PROGRAM CheckConfig
VAR_INPUT
		IN_Start				: BOOL := TRUE;
		ParamInitWait			: TIME := T#5S;
END_VAR
VAR_OUTPUT
		OUT_aDBConfig         		: ARRAY[0..MAX_CONFIGURATIONS] OF ST_ConfigDB;
		OUT_Busy					: BOOL;
		OUT_Error					: BOOL;
		OUT_Result					: INT;
END_VAR
VAR
	// CheckConfig    
		TON_CheckConfig				: TON;      		
		TrigCheckConfig				: R_TRIG;
		TrigInit					: F_TRIG;
		RS_CheckConfig				: RS;
		                    		
		ConfigTcDBSrvEvt  			: FB_ConfigTcDBSrvEvt(sNetId := '', tTimeout:=T#5S);
		                    		
		aAutoGrpConfig    			: ARRAY[0..MAX_CONFIGURATIONS] OF ST_ConfigAutoLogGrp;
		AX_NameBase					: ARRAY[0..MAX_CONFIGURATIONS] OF T_MaxString;
		AX_hDBID					: ARRAY[0..MAX_CONFIGURATIONS] OF BOOL;
		AX_hDBIDNull				: ARRAY[0..MAX_CONFIGURATIONS] OF BOOL;
		                    		
		nDbCount          			: UDINT;
		nAutoGrpCount     			: UDINT;

		KK : UDINT;
END_VAR

TON_CheckConfig(IN := IN_Start, PT := ParamInitWait);

TrigCheckConfig(CLK := TON_CheckConfig.Q);
RS_CheckConfig(SET := TrigCheckConfig.Q);
IF TrigCheckConfig.Q THEN
	IN_Start := FALSE;
	OUT_Result := 0;
END_IF
IF RS_CheckConfig.Q1 THEN
	
	OUT_Busy := TRUE;
	IF ConfigTcDBSrvEvt.Read(pDBConfig := ADR(OUT_aDBConfig), cbDBConfig := SIZEOF(OUT_aDBConfig), pAutologGrpConfig := ADR(aAutoGrpConfig),
			cbAutoLogGrpConfig := SIZEOF(aAutoGrpConfig),pDBCount := ADR(nDbCount),pAutoLogGrpCount := ADR(nAutoGrpCount)) THEN
		
		IF ConfigTcDBSrvEvt.bError THEN
			OUT_Result := -1;
		ELSE
			FOR KK := 0 TO MAX_CONFIGURATIONS DO
				AX_hDBID[OUT_aDBConfig[KK].hDBID] := OUT_aDBConfig[KK].hDBID <> 0;
				AX_NameBase[KK] :=  OUT_aDBConfig[KK].sName;
			END_FOR
			OUT_Result := 1;
		END_IF  
		RS_CheckConfig(RESET1 := TRUE);
		RS_CheckConfig(RESET1 := FALSE);
		OUT_Busy := FALSE;
		
	END_IF
END_IF

END_PROGRAM

(* stored: Version 1.1.0.1, ProductVersion 3.1.4024.6
   POU CheckConfig: Id {503db43f-1be2-4b73-b610-623c8286b0be}, SpecialFunc None *)
